FUNCTION_BLOCK {BlockName}_HMI
  PACKAGE {YourNamespace};
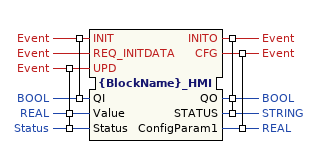
  EVENT_INPUT
    INIT WITH QI;
    REQ_INITDATA;
    UPD WITH Value, Status;
  END_EVENT
  EVENT_OUTPUT
    INITO WITH QO, STATUS;
    CFG WITH ConfigParam1;
  END_EVENT
  VAR_INPUT
    QI : BOOL;
    Value : REAL;
    Status : Status;
  END_VAR
  VAR_OUTPUT
    QO : BOOL;
    STATUS : STRING;
    ConfigParam1 : REAL;
  END_VAR
  SERVICE /
    SEQUENCE 
    END_SEQUENCE
  END_SERVICE
END_FUNCTION_BLOCK
